// TIA Portal V17 export
// export: Created 2023-06-23T18:33:39.7522261Z, ExportSetting WithDefaults, DisplayName Totally Integrated Automation Portal, DisplayVersion V17, DisplayName TIA Portal Openness, DisplayVersion V17, DisplayName TIA Portal Version Control Interface, DisplayVersion V17, DisplayName STEP 7 Professional, DisplayVersion V17, DisplayName STEP 7 Safety, DisplayVersion V17, DisplayName WinCC Advanced / Unified PC, DisplayVersion V17
VAR_GLOBAL   // PLC tag table "18_AE2-SA2"
   "iAE2-SA2p" AT %I9.6 : Bool;   // 7
   "iAE2-SA2" AT %I9.7 : Bool;   // 7
   "iAE2-SA2a" AT %I17.5 : Bool;
   "oAE2-SA2p" AT %Q9.1 : Bool;
   "oAE2-SA2" AT %Q9.2 : Bool;
END_VAR
